(* IEC 61131-3 sources: moqui-plc/iec61131/moqui/framework/src/main/org/moqui/util, 39 files *)

(* ---- Clocks.dut ---- *)
(*#-#-#-#-#-#-#-#-#-#---Declaration---#-#-#-#-#-#-#-#-#-#-#-#-#*)

(* Generated clocks for timing generation *)
TYPE Clocks : STRUCT
	(*
     * SystemClock is the main high-speed clock, e.g., from the task cycle.
     * All other clocks are derived from it.
     *)
    systemClock : BOOL; (* Main system clock 100 Hz, duty-cycle 50% *)
    (* Derived clock pulses (one-cycle TRUE). Derived from systemClock rising edge *)
    clock10ms : BOOL; (* 10ms pulse *)
    clock100ms : BOOL; (* 100ms pulse *)
    clock1s : BOOL; (* 1 second pulse *)
    clock1minute : BOOL; (* 1 minute pulse *)
	(* Extend based on your needs *)
END_STRUCT END_TYPE

(* ---- Clocks.st ---- *)
(* Generated clocks for timing generation *)
TYPE Clocks : STRUCT
	(*
     * SystemClock is the main high-speed clock, e.g., from the task cycle.
     * All other clocks are derived from it.
     *)
    systemClock : BOOL; (* Main system clock 100 Hz, duty-cycle 50% *)
    (* Derived clock pulses (one-cycle TRUE). Derived from systemClock rising edge *)
    clock10ms : BOOL; (* 10ms pulse *)
    clock100ms : BOOL; (* 100ms pulse *)
    clock1s : BOOL; (* 1 second pulse *)
    clock1minute : BOOL; (* 1 minute pulse *)
	(* Extend based on your needs *)
END_STRUCT END_TYPE

(* ---- MeanFilterType.dut ---- *)
(*#-#-#-#-#-#-#-#-#-#---Declaration---#-#-#-#-#-#-#-#-#-#-#-#-#*)

{attribute 'qualified_only'}
{attribute 'strict'}
TYPE MeanFilterType : (
    SMA, (* Simple Moving Average *)
    WMA_Ramp, (* Weighted Moving Average, linear weights 1..N from oldest..newest (O(1)) *)
    WMA_Triangular, (* Symmetric triangular weights, center-weighted (O(N)) *)
    WMA_TriangularOddOnly, (* Symmetric triangular weights, requires odd windowSize (O(N)) *)
    TRI_SMA2, (* Triangular approximation via two SMA in cascade (O(1) per tick, extra memory) *)
    EMA (* Exponential Moving Average (alpha mandatory) *)
); END_TYPE

(* ---- doubleWordToReal.pou ---- *)
(*#-#-#-#-#-#-#-#-#-#---Declaration---#-#-#-#-#-#-#-#-#-#-#-#-#*)

(* Utility function to convert a word array to a real variable *)
FUNCTION doubleWordToReal : REAL
VAR_INPUT
	wordArray : ARRAY[0..1] OF WORD;
	bigEndian : BOOL := FALSE;
END_VAR
VAR
    dwordValue : DWORD;
END_VAR

(*#-#-#-#-#-#-#-#-#-#---Implementation---#-#-#-#-#-#-#-#-#-#-#-#-#*)

dwordValue := SHL(TO_DWORD(wordArray[0]), 16) OR TO_DWORD(wordArray[1]);
IF bigEndian THEN
    dwordValue := swapDWordEndian(dwordValue);
END_IF;
doubleWordToReal := TO_REAL(dwordValue);

(* ---- doubleWordToReal.st ---- *)
(* Utility function to convert a word array to a real variable *)
FUNCTION doubleWordToReal : REAL
	VAR_INPUT
		wordArray : ARRAY[0..1] OF WORD;
		bigEndian : BOOL := FALSE;
	END_VAR
	VAR
	    dwordValue : DWORD;
	END_VAR

	dwordValue := SHL(TO_DWORD(wordArray[0]), 16) OR TO_DWORD(wordArray[1]);
	IF bigEndian THEN
	    dwordValue := swapDWordEndian(dwordValue);
	END_IF;
	doubleWordToReal := TO_REAL(dwordValue);
	END_FUNCTION

(* ---- longRealToWordArray.pou ---- *)
(*#-#-#-#-#-#-#-#-#-#---Declaration---#-#-#-#-#-#-#-#-#-#-#-#-#*)

(* Convert a long real variable to a word array *)
FUNCTION longRealToWordArray : ARRAY[0..3] OF WORD
VAR_INPUT
    value : LREAL;
    bigEndian : BOOL := FALSE;
END_VAR
VAR
    lwordValue : LWORD;
    result : ARRAY[0..3] OF WORD;
END_VAR

(*#-#-#-#-#-#-#-#-#-#---Implementation---#-#-#-#-#-#-#-#-#-#-#-#-#*)

lwordValue := TO_LWORD(value);
IF bigEndian THEN
    lwordValue := swapLWordEndian(lwordValue);
END_IF;

result[0] := TO_WORD(SHR(lwordValue, 48));
result[1] := TO_WORD(SHR(lwordValue, 32) AND 16#FFFF);
result[2] := TO_WORD(SHR(lwordValue, 16) AND 16#FFFF);
result[3] := TO_WORD(lwordValue AND 16#FFFF);
longRealToWordArray := result;

(* ---- longRealToWordArray.st ---- *)
(* Convert a long real variable to a word array *)
FUNCTION longRealToWordArray : ARRAY[0..3] OF WORD
	VAR_INPUT
	    value : LREAL;
	    bigEndian : BOOL := FALSE;
	END_VAR
	VAR
	    lwordValue : LWORD;
	    result : ARRAY[0..3] OF WORD;
	END_VAR

	lwordValue := TO_LWORD(value);
	IF bigEndian THEN
	    lwordValue := swapLWordEndian(lwordValue);
	END_IF;

	result[0] := TO_WORD(SHR(lwordValue, 48));
	result[1] := TO_WORD(SHR(lwordValue, 32) AND 16#FFFF);
	result[2] := TO_WORD(SHR(lwordValue, 16) AND 16#FFFF);
	result[3] := TO_WORD(lwordValue AND 16#FFFF);
	longRealToWordArray := result;
	END_FUNCTION

(* ---- longWordToLongReal.pou ---- *)
(*#-#-#-#-#-#-#-#-#-#---Declaration---#-#-#-#-#-#-#-#-#-#-#-#-#*)

(* Utility function to convert a word array to a long real variable *)
FUNCTION longWordToLongReal : LREAL
VAR_INPUT
	wordArray : ARRAY[0..3] OF WORD;
	bigEndian : BOOL := FALSE;
END_VAR
VAR
	lwordValue : LWORD;
	w : ARRAY[0..3] OF WORD;
END_VAR

(*#-#-#-#-#-#-#-#-#-#---Implementation---#-#-#-#-#-#-#-#-#-#-#-#-#*)

IF bigEndian THEN
    w[0] := wordArray[3];
    w[1] := wordArray[2];
    w[2] := wordArray[1];
    w[3] := wordArray[0];
ELSE
    w := wordArray;
END_IF;

lwordValue := TO_LWORD(w[3]);
lwordValue := SHL(lwordValue, 16) OR TO_LWORD(w[2]);
lwordValue := SHL(lwordValue, 16) OR TO_LWORD(w[1]);
lwordValue := SHL(lwordValue, 16) OR TO_LWORD(w[0]);
longWordToLongReal := TO_LREAL(lwordValue);

(* ---- longWordToLongReal.st ---- *)
(* Utility function to convert a word array to a long real variable *)
FUNCTION longWordToLongReal : LREAL
	VAR_INPUT
		wordArray : ARRAY[0..3] OF WORD;
		bigEndian : BOOL := FALSE;
	END_VAR
	VAR
		lwordValue : LWORD;
		w : ARRAY[0..3] OF WORD;
	END_VAR

	IF bigEndian THEN
	    w[0] := wordArray[3];
	    w[1] := wordArray[2];
	    w[2] := wordArray[1];
	    w[3] := wordArray[0];
	ELSE
	    w := wordArray;
	END_IF;

	lwordValue := TO_LWORD(w[3]);
	lwordValue := SHL(lwordValue, 16) OR TO_LWORD(w[2]);
	lwordValue := SHL(lwordValue, 16) OR TO_LWORD(w[1]);
	lwordValue := SHL(lwordValue, 16) OR TO_LWORD(w[0]);
	longWordToLongReal := TO_LREAL(lwordValue);
	END_FUNCTION

(* ---- nowTimestamp.pou ---- *)
(*#-#-#-#-#-#-#-#-#-#---Declaration---#-#-#-#-#-#-#-#-#-#-#-#-#*)

FUNCTION nowTimestamp : DATE_AND_TIME
VAR
    utcTimestamp: UDINT;
    localTimestamp: UDINT;
    result: SysTimeRtc.RTS_IEC_RESULT;
	nowTimestampLocalString : STRING;
END_VAR

(*#-#-#-#-#-#-#-#-#-#---Implementation---#-#-#-#-#-#-#-#-#-#-#-#-#*)

(* Get current UTC time *)
utcTimestamp := SysTimeRtcGet(result);
(* Handle error (log it, return a default timestamp, etc.) *)
IF result <> 0 THEN RETURN; END_IF;
(* Convert UTC seconds to local time *)
result := SysTimeRtcConvertUtcToLocal(utcTimestamp, localTimestamp);
IF result <> 0 THEN RETURN; END_IF;
(* Convert local time to data and time format *)
nowTimestamp := TO_DT(localTimestamp);
(* Convert date and time format to a string *)
nowTimestampLocalString := TO_STRING(nowTimestamp);

(* ---- nowTimestamp.st ---- *)
FUNCTION nowTimestamp : DATE_AND_TIME
	VAR
	    utcTimestamp: UDINT;
	    localTimestamp: UDINT;
	    result: SysTimeRtc.RTS_IEC_RESULT;
		nowTimestampLocalString : STRING;
	END_VAR

	(* Get current UTC time *)
	utcTimestamp := SysTimeRtcGet(result);
	(* Handle error (log it, return a default timestamp, etc.) *)
	IF result <> 0 THEN RETURN; END_IF;
	(* Convert UTC seconds to local time *)
	result := SysTimeRtcConvertUtcToLocal(utcTimestamp, localTimestamp);
	IF result <> 0 THEN RETURN; END_IF;
	(* Convert local time to data and time format *)
	nowTimestamp := TO_DT(localTimestamp);
	(* Convert date and time format to a string *)
	nowTimestampLocalString := TO_STRING(nowTimestamp);
	END_FUNCTION

(* ---- realToWordArray.pou ---- *)
(*#-#-#-#-#-#-#-#-#-#---Declaration---#-#-#-#-#-#-#-#-#-#-#-#-#*)

(* Convert a real variable to a word array *)
FUNCTION realToWordArray : ARRAY[0..1] OF WORD
VAR_INPUT
    value : REAL;
    bigEndian : BOOL := FALSE;
END_VAR
VAR
    dwordValue : DWORD;
    result : ARRAY[0..1] OF WORD;
END_VAR

(*#-#-#-#-#-#-#-#-#-#---Implementation---#-#-#-#-#-#-#-#-#-#-#-#-#*)

dwordValue := TO_DWORD(value);
IF bigEndian THEN
    dwordValue := swapDWordEndian(dwordValue);
END_IF;
result[0] := TO_WORD(SHR(dwordValue, 16));
result[1] := TO_WORD(dwordValue AND 16#FFFF);
realToWordArray := result;

(* ---- realToWordArray.st ---- *)
(* Convert a real variable to a word array *)
FUNCTION realToWordArray : ARRAY[0..1] OF WORD
	VAR_INPUT
	    value : REAL;
	    bigEndian : BOOL := FALSE;
	END_VAR
	VAR
	    dwordValue : DWORD;
	    result : ARRAY[0..1] OF WORD;
	END_VAR

	dwordValue := TO_DWORD(value);
	IF bigEndian THEN
	    dwordValue := swapDWordEndian(dwordValue);
	END_IF;
	result[0] := TO_WORD(SHR(dwordValue, 16));
	result[1] := TO_WORD(dwordValue AND 16#FFFF);
	realToWordArray := result;
	END_FUNCTION

(* ---- round.pou ---- *)
(*#-#-#-#-#-#-#-#-#-#---Declaration---#-#-#-#-#-#-#-#-#-#-#-#-#*)

FUNCTION round : REAL
VAR_INPUT
    inputValue : REAL;
    decimals : INT;
END_VAR
VAR
    factor : REAL;
    tempValue : REAL;
END_VAR

(*#-#-#-#-#-#-#-#-#-#---Implementation---#-#-#-#-#-#-#-#-#-#-#-#-#*)

factor := TO_REAL(EXP(LN(10.0) * decimals));
tempValue := inputValue * factor;

IF tempValue >= 0 THEN
    round := TO_REAL(TRUNC(tempValue + 0.5)) / factor;
ELSE
    round := TO_REAL(TRUNC(tempValue - 0.5)) / factor;
END_IF;

(* ---- round.st ---- *)
FUNCTION round : REAL
	VAR_INPUT
	    inputValue : REAL;
	    decimals : INT;
	END_VAR
	VAR
	    factor : REAL;
	    tempValue : REAL;
	END_VAR

	factor := TO_REAL(EXP(LN(10.0) * decimals));
	tempValue := inputValue * factor;

	IF tempValue >= 0 THEN
	    round := TO_REAL(TRUNC(tempValue + 0.5)) / factor;
	ELSE
	    round := TO_REAL(TRUNC(tempValue - 0.5)) / factor;
	END_IF;
	END_FUNCTION

(* ---- scale.pou ---- *)
(*#-#-#-#-#-#-#-#-#-#---Declaration---#-#-#-#-#-#-#-#-#-#-#-#-#*)

FUNCTION scale : REAL
VAR_INPUT
	inputValue: REAL;
	minInputValue: REAL;
	maxInputValue: REAL;
	minOutputValue: REAL;
	maxOutputValue: REAL;
END_VAR
VAR
	outputValue: REAL;
END_VAR

(*#-#-#-#-#-#-#-#-#-#---Implementation---#-#-#-#-#-#-#-#-#-#-#-#-#*)

IF maxInputValue <= minInputValue THEN
	outputValue := minOutputValue;
ELSE
    outputValue := (maxOutputValue - minOutputValue) / (maxInputValue - minInputValue)
		* (LIMIT(minInputValue, inputValue, maxInputValue) - minInputValue) + minOutputValue;
END_IF;
scale := outputValue;

(* ---- scale.st ---- *)
FUNCTION scale : REAL
	VAR_INPUT
		inputValue: REAL;
		minInputValue: REAL;
		maxInputValue: REAL;
		minOutputValue: REAL;
		maxOutputValue: REAL;
	END_VAR
	VAR
		outputValue: REAL;
	END_VAR

	IF maxInputValue <= minInputValue THEN
		outputValue := minOutputValue;
	ELSE
	    outputValue := (maxOutputValue - minOutputValue) / (maxInputValue - minInputValue)
			* (LIMIT(minInputValue, inputValue, maxInputValue) - minInputValue) + minOutputValue;
	END_IF;
	scale := outputValue;
	END_FUNCTION

(* ---- swapDWordEndian.pou ---- *)
(*#-#-#-#-#-#-#-#-#-#---Declaration---#-#-#-#-#-#-#-#-#-#-#-#-#*)

(* Swap two words in a double word to change the endianness *)
FUNCTION swapDWordEndian : DWORD
VAR_INPUT
    input : DWORD;
END_VAR

(*#-#-#-#-#-#-#-#-#-#---Implementation---#-#-#-#-#-#-#-#-#-#-#-#-#*)

swapDWordEndian := SHL(input AND 16#0000FFFF, 16) OR SHR(input AND 16#FFFF0000, 16);

(* ---- swapDWordEndian.st ---- *)
(* Swap two words in a double word to change the endianness *)
FUNCTION swapDWordEndian : DWORD
	VAR_INPUT
	    input : DWORD;
	END_VAR

	swapDWordEndian := SHL(input AND 16#0000FFFF, 16) OR SHR(input AND 16#FFFF0000, 16);
	END_FUNCTION

(* ---- swapLWordEndian.pou ---- *)
(*#-#-#-#-#-#-#-#-#-#---Declaration---#-#-#-#-#-#-#-#-#-#-#-#-#*)

(* Swap four words in an long word *)
FUNCTION swapLWordEndian : LWORD
VAR_INPUT
    input : LWORD;
END_VAR
VAR
    w0, w1, w2, w3 : WORD;
    result : LWORD;
END_VAR

(*#-#-#-#-#-#-#-#-#-#---Implementation---#-#-#-#-#-#-#-#-#-#-#-#-#*)

w0 := TO_WORD(SHR(input, 48));
w1 := TO_WORD(SHR(input, 32) AND 16#FFFF);
w2 := TO_WORD(SHR(input, 16) AND 16#FFFF);
w3 := TO_WORD(input AND 16#FFFF);
result := TO_LWORD(w3);
result := SHL(result, 16) OR TO_LWORD(w2);
result := SHL(result, 16) OR TO_LWORD(w1);
result := SHL(result, 16) OR TO_LWORD(w0);
swapLWordEndian := result;

(* ---- swapLWordEndian.st ---- *)
(* Swap four words in an long word *)
FUNCTION swapLWordEndian : LWORD
	VAR_INPUT
	    input : LWORD;
	END_VAR
	VAR
	    w0, w1, w2, w3 : WORD;
	    result : LWORD;
	END_VAR

	w0 := TO_WORD(SHR(input, 48));
	w1 := TO_WORD(SHR(input, 32) AND 16#FFFF);
	w2 := TO_WORD(SHR(input, 16) AND 16#FFFF);
	w3 := TO_WORD(input AND 16#FFFF);
	result := TO_LWORD(w3);
	result := SHL(result, 16) OR TO_LWORD(w2);
	result := SHL(result, 16) OR TO_LWORD(w1);
	result := SHL(result, 16) OR TO_LWORD(w0);
	swapLWordEndian := result;
	END_FUNCTION

(* ---- swapWordEndian.pou ---- *)
(*#-#-#-#-#-#-#-#-#-#---Declaration---#-#-#-#-#-#-#-#-#-#-#-#-#*)

(* Swap bytes in a word to change the endianness *)
FUNCTION swapWordEndian : WORD
VAR_INPUT
    input : WORD;
END_VAR

(*#-#-#-#-#-#-#-#-#-#---Implementation---#-#-#-#-#-#-#-#-#-#-#-#-#*)

swapWordEndian := SHL(input AND 16#00FF, 8) OR SHR(input AND 16#FF00, 8);

(* ---- swapWordEndian.st ---- *)
(* Swap bytes in a word to change the endianness *)
FUNCTION swapWordEndian : WORD
	VAR_INPUT
	    input : WORD;
	END_VAR

	swapWordEndian := SHL(input AND 16#00FF, 8) OR SHR(input AND 16#FF00, 8);
	END_FUNCTION

(* ---- toByteArray.pou ---- *)
(*#-#-#-#-#-#-#-#-#-#---Declaration---#-#-#-#-#-#-#-#-#-#-#-#-#*)

FUNCTION toByteArray : BOOL
VAR_INPUT
    inputWord : WORD;
END_VAR
VAR_OUTPUT
	byteArray : ARRAY [0..1] OF BYTE; (* Output array: [highByte, lowByte] *)
END_VAR

(*#-#-#-#-#-#-#-#-#-#---Implementation---#-#-#-#-#-#-#-#-#-#-#-#-#*)

toByteArray := FALSE;
(* Extract high and low byte *)
byteArray[0] := TO_BYTE(SHR(inputWord, 8)); (* High byte *)
byteArray[1] := TO_BYTE(inputWord AND 16#00FF); (* Low byte *)
toByteArray := TRUE;

(* ---- toByteArray.st ---- *)
FUNCTION toByteArray : BOOL
	VAR_INPUT
	    inputWord : WORD;
	END_VAR
	VAR_OUTPUT
		byteArray : ARRAY [0..1] OF BYTE; (* Output array: [highByte, lowByte] *)
	END_VAR

	toByteArray := FALSE;
	(* Extract high and low byte *)
	byteArray[0] := TO_BYTE(SHR(inputWord, 8)); (* High byte *)
	byteArray[1] := TO_BYTE(inputWord AND 16#00FF); (* Low byte *)
	toByteArray := TRUE;
	END_FUNCTION

(* ---- trim.pou ---- *)
(*#-#-#-#-#-#-#-#-#-#---Declaration---#-#-#-#-#-#-#-#-#-#-#-#-#*)

FUNCTION trim : STRING
VAR_INPUT
    inputString : STRING;
END_VAR
VAR
    startPos, endPos : INT;
    stringLength : INT;
    currentCharCode : INT;
END_VAR

(*#-#-#-#-#-#-#-#-#-#---Implementation---#-#-#-#-#-#-#-#-#-#-#-#-#*)

stringLength := LEN(inputString);
startPos := 1;

(* Skip leading whitespace (space, tab = 9, LF = 10, CR = 13) *)
WHILE (startPos <= stringLength) DO
    currentCharCode := TO_INT(MID(inputString, startPos, 1));
    IF (currentCharCode <> 32) AND (currentCharCode <> 9)
			AND (currentCharCode <> 10) AND (currentCharCode <> 13) THEN
        EXIT;
    END_IF;

    startPos := startPos + 1;
END_WHILE;

(* Skip trailing whitespace *)
endPos := stringLength;
WHILE (endPos > 0) DO
    currentCharCode := TO_INT(MID(inputString, endPos, 1));
    IF (currentCharCode <> 32) AND (currentCharCode <> 9)
			AND (currentCharCode <> 10) AND (currentCharCode <> 13) THEN
        EXIT;
    END_IF;

    endPos := endPos - 1;
END_WHILE;

(* Extract the trimmed substring *)
IF startPos <= endPos THEN
    trim := MID(inputString, startPos, endPos - startPos + 1);
ELSE
    trim := ''; (* All characters were whitespace *)
END_IF;

(* ---- trim.st ---- *)
FUNCTION trim : STRING
	VAR_INPUT
	    inputString : STRING;
	END_VAR
	VAR
	    startPos, endPos : INT;
	    stringLength : INT;
	    currentCharCode : INT;
	END_VAR

	stringLength := LEN(inputString);
	startPos := 1;

	(* Skip leading whitespace (space, tab = 9, LF = 10, CR = 13) *)
	WHILE (startPos <= stringLength) DO
	    currentCharCode := TO_INT(MID(inputString, startPos, 1));
	    IF (currentCharCode <> 32) AND (currentCharCode <> 9)
				AND (currentCharCode <> 10) AND (currentCharCode <> 13) THEN
	        EXIT;
	    END_IF;

	    startPos := startPos + 1;
	END_WHILE;

	(* Skip trailing whitespace *)
	endPos := stringLength;
	WHILE (endPos > 0) DO
	    currentCharCode := TO_INT(MID(inputString, endPos, 1));
	    IF (currentCharCode <> 32) AND (currentCharCode <> 9)
				AND (currentCharCode <> 10) AND (currentCharCode <> 13) THEN
	        EXIT;
	    END_IF;

	    endPos := endPos - 1;
	END_WHILE;

	(* Extract the trimmed substring *)
	IF startPos <= endPos THEN
	    trim := MID(inputString, startPos, endPos - startPos + 1);
	ELSE
	    trim := ''; (* All characters were whitespace *)
	END_IF;
	END_FUNCTION

(* ---- truncReal.pou ---- *)
(*#-#-#-#-#-#-#-#-#-#---Declaration---#-#-#-#-#-#-#-#-#-#-#-#-#*)

FUNCTION truncReal : REAL
VAR_INPUT
    inputValue : REAL;
    decimals : INT;
END_VAR
VAR
    factor : REAL;
END_VAR

(*#-#-#-#-#-#-#-#-#-#---Implementation---#-#-#-#-#-#-#-#-#-#-#-#-#*)

factor := TO_REAL(EXP(LN(10.0) * TO_REAL(decimals)));
truncReal := TO_REAL(TRUNC(inputValue * factor)) / factor;

(* ---- truncReal.st ---- *)
FUNCTION truncReal : REAL
	VAR_INPUT
	    inputValue : REAL;
	    decimals : INT;
	END_VAR
	VAR
	    factor : REAL;
	END_VAR

	factor := TO_REAL(EXP(LN(10.0) * TO_REAL(decimals)));
	truncReal := TO_REAL(TRUNC(inputValue * factor)) / factor;
	END_FUNCTION

(* ---- ClockGeneration.pou ---- *)
(*#-#-#-#-#-#-#-#-#-#---Declaration---#-#-#-#-#-#-#-#-#-#-#-#-#*)

{attribute 'no_assign'}
(* Timing generation *)
FUNCTION_BLOCK ClockGeneration
VAR_EXTERNAL
	clks : Clocks;
END_VAR
VAR_INPUT
	operationType : OperatingMode;
END_VAR
VAR
	(* Internal variable to detect the rising edge of the systemClock *)
	systemClockOld : BOOL;
	(* Internal counters for derived clocks *)
	timerClock100ms : UDINT;
	timerClock1s : UDINT;
	timerClock1minute : UDINT;
END_VAR

(*#-#-#-#-#-#-#-#-#-#---Implementation---#-#-#-#-#-#-#-#-#-#-#-#-#*)

IF (operationType = OperatingMode.Init) THEN
	systemClockOld := TRUE;
	timerClock100ms := 10;
	timerClock1s := 10;
	timerClock1minute := 60;
END_IF;

(*
 * Uncomment if you want to make loops shorter than 10 ms.
 * It is not recommended to go below 5 ms with the PLC.
 * The control loop (current) of the axes is in the servo drives.
 *)
(*
clks.clock10ms := clks.systemClock AND NOT systemClockOld;
systemClockOld := clks.systemClock;
*)
clks.clock10ms := TRUE;

IF clks.clock10ms THEN
	timerClock100ms := timerClock100ms - 1;
END_IF;
clks.clock100ms := (timerClock100ms = 0);

IF clks.clock100ms THEN
	timerClock100ms := 10;
	timerClock1s := timerClock1s - 1;
END_IF;
clks.clock1s := (timerClock1s = 0);

IF clks.clock1s THEN
	timerClock1s := 10;
	timerClock1minute := timerClock1minute - 1;
END_IF;
clks.clock1minute := (timerClock1minute = 0);

IF clks.clock1minute THEN
	timerClock1minute := 60;
END_IF;

(* ---- ClockGeneration.st ---- *)
(* Timing generation *)
FUNCTION_BLOCK ClockGeneration
	VAR_EXTERNAL
		clks : Clocks;
	END_VAR
	VAR_INPUT
		operationType : OperatingMode;
	END_VAR
	VAR
		(* Internal variable to detect the rising edge of the systemClock *)
		systemClockOld : BOOL;
		(* Internal counters for derived clocks *)
		timerClock100ms : UDINT;
		timerClock1s : UDINT;
		timerClock1minute : UDINT;
	END_VAR

	IF (operationType = OperatingMode.Init) THEN
		systemClockOld := TRUE;
		timerClock100ms := 10;
		timerClock1s := 10;
		timerClock1minute := 60;
	END_IF;

	(*
	 * Uncomment if you want to make loops shorter than 10 ms.
	 * It is not recommended to go below 5 ms with the PLC.
	 * The control loop (current) of the axes is in the servo drives.
	 *)
	(*
	clks.clock10ms := clks.systemClock AND NOT systemClockOld;
	systemClockOld := clks.systemClock;
	*)
	clks.clock10ms := TRUE;

	IF clks.clock10ms THEN
		timerClock100ms := timerClock100ms - 1;
	END_IF;
	clks.clock100ms := (timerClock100ms = 0);

	IF clks.clock100ms THEN
		timerClock100ms := 10;
		timerClock1s := timerClock1s - 1;
	END_IF;
	clks.clock1s := (timerClock1s = 0);

	IF clks.clock1s THEN
		timerClock1s := 10;
		timerClock1minute := timerClock1minute - 1;
	END_IF;
	clks.clock1minute := (timerClock1minute = 0);

	IF clks.clock1minute THEN
		timerClock1minute := 60;
	END_IF;
	END_FUNCTION_BLOCK

(* ---- Filter.pou ---- *)
(*#-#-#-#-#-#-#-#-#-#---Declaration---#-#-#-#-#-#-#-#-#-#-#-#-#*)

(* Signal filtering and deboucing.
   Usage:

       (* heatingPlatesOpened *)
       VAR
           heatingPlatesOpenedFilter : Filter;
       END_VAR

       heatingPlatesOpenedFilter(operationType := operationType, clock := heatingPlatesControlClock,
           signal := heatingPlatesOpened, activationDelay := 0, deactivationDelay := heatingPlatesOpeningDelay,
	   	   delayedSignal => heatingPlatesOpened);
 *)
FUNCTION_BLOCK Filter
VAR_INPUT
	operationType : OperatingMode;
	clock : BOOL;
	signal : BOOL;
	activationDelay : UDINT;
	deactivationDelay : UDINT;
END_VAR
VAR_OUTPUT
	delayedSignal : BOOL;
END_VAR
VAR
	delay : UDINT;
END_VAR

(*#-#-#-#-#-#-#-#-#-#---Implementation---#-#-#-#-#-#-#-#-#-#-#-#-#*)

IF (operationType = OperatingMode.Init) THEN
	delay := 0;
END_IF;

IF clock AND (delay > 0) THEN
	delay := delay - 1;
END_IF;

IF delay = 0 THEN
	delayedSignal := signal;
END_IF;

IF signal = delayedSignal THEN
	IF signal THEN
		delay := deactivationDelay;
	ELSE
		delay := activationDelay;
	END_IF;
END_IF;

(* ---- Filter.st ---- *)
(* Signal filtering and deboucing.
   Usage:

       (* heatingPlatesOpened *)
       VAR
           heatingPlatesOpenedFilter : Filter;
       END_VAR

       heatingPlatesOpenedFilter(operationType := operationType, clock := heatingPlatesControlClock,
           signal := heatingPlatesOpened, activationDelay := 0, deactivationDelay := heatingPlatesOpeningDelay,
	   	   delayedSignal => heatingPlatesOpened);
 *)
FUNCTION_BLOCK Filter
VAR_INPUT
	operationType : OperatingMode;
	clock : BOOL;
	signal : BOOL;
	activationDelay : UDINT;
	deactivationDelay : UDINT;
END_VAR
VAR_OUTPUT
	delayedSignal : BOOL;
END_VAR
VAR
	delay : UDINT;
END_VAR

IF (operationType = OperatingMode.Init) THEN
	delay := 0;
END_IF;

IF clock AND (delay > 0) THEN
	delay := delay - 1;
END_IF;

IF delay = 0 THEN
	delayedSignal := signal;
END_IF;

IF signal = delayedSignal THEN
	IF signal THEN
		delay := deactivationDelay;
	ELSE
		delay := activationDelay;
	END_IF;
END_IF;

(* ---- IIRFilter.pou ---- *)
(*#-#-#-#-#-#-#-#-#-#---Declaration---#-#-#-#-#-#-#-#-#-#-#-#-#*)

{attribute 'no_assign'}
FUNCTION_BLOCK IIRFilter
VAR_INPUT
    execute : BOOL;
    clock : BOOL;
    reset : BOOL;
    input : REAL;
    T : REAL; (* Time constant in seconds *)
    tickTime : TIME := T#10ms; (* Sampling period *)
END_VAR
VAR_OUTPUT
    output : REAL;
    done : BOOL;
    busy : BOOL;
    error : BOOL;
    errorId : INT; (* 1 : InvalidTime *)
    timeElapsed : REAL; (* Time elapsed in seconds *)
END_VAR
VAR
    init : BOOL;
    elapsedTicks : UDINT;
    deltaTime : REAL;
    alpha : REAL;
END_VAR

(*#-#-#-#-#-#-#-#-#-#---Implementation---#-#-#-#-#-#-#-#-#-#-#-#-#*)

(* Defaults *)
done := FALSE; busy := FALSE; error := FALSE; errorId := 0;

(* Validate tickTime *)
IF TO_DINT(tickTime) <= 0 THEN
    error := execute;
    errorId := 1;
    busy := FALSE;
    RETURN;
END_IF;

deltaTime := TO_REAL(TO_DINT(tickTime)) / 1000.0; (* seconds per tick *)

IF reset THEN
    init := FALSE;
    elapsedTicks := 0;
END_IF;

IF execute THEN
    busy := TRUE;

    (* Initialize output to current input on first enable *)
    IF NOT init THEN
        output := input;
        init := TRUE;
        elapsedTicks := 0;
    ELSE
        (* Update only on external tick *)
        IF clock THEN
            (* alpha = 1 - exp(-dt/T) *)
            IF T > 0.0 THEN
                alpha := 1.0 - EXP(-deltaTime / T);
                output := output + alpha * (input - output);
            ELSE
                output := input;
            END_IF;

            elapsedTicks := elapsedTicks + 1;
        END_IF;
    END_IF;

    timeElapsed := TO_REAL(elapsedTicks) * deltaTime;

    done := NOT error;
ELSE
    busy := FALSE;
    done := FALSE;
    timeElapsed := 0.0;
END_IF;

(* ---- IIRFilter.st ---- *)
FUNCTION_BLOCK IIRFilter
	VAR_INPUT
	    execute : BOOL;
	    clock : BOOL;
	    reset : BOOL;
	    input : REAL;
	    T : REAL; (* Time constant in seconds *)
	    tickTime : TIME := T#10ms; (* Sampling period *)
	END_VAR
	VAR_OUTPUT
	    output : REAL;
	    done : BOOL;
	    busy : BOOL;
	    error : BOOL;
	    errorId : INT; (* 1 : InvalidTime *)
	    timeElapsed : REAL; (* Time elapsed in seconds *)
	END_VAR
	VAR
	    init : BOOL;
	    elapsedTicks : UDINT;
	    deltaTime : REAL;
	    alpha : REAL;
	END_VAR

	(* Defaults *)
	done := FALSE; busy := FALSE; error := FALSE; errorId := 0;

	(* Validate tickTime *)
	IF TO_DINT(tickTime) <= 0 THEN
	    error := execute;
	    errorId := 1;
	    busy := FALSE;
	    RETURN;
	END_IF;

	deltaTime := TO_REAL(TO_DINT(tickTime)) / 1000.0; (* seconds per tick *)

	IF reset THEN
	    init := FALSE;
	    elapsedTicks := 0;
	END_IF;

	IF execute THEN
	    busy := TRUE;

	    (* Initialize output to current input on first enable *)
	    IF NOT init THEN
	        output := input;
	        init := TRUE;
	        elapsedTicks := 0;
	    ELSE
	        (* Update only on external tick *)
	        IF clock THEN
	            (* alpha = 1 - exp(-dt/T) *)
	            IF T > 0.0 THEN
	                alpha := 1.0 - EXP(-deltaTime / T);
	                output := output + alpha * (input - output);
	            ELSE
	                output := input;
	            END_IF;

	            elapsedTicks := elapsedTicks + 1;
	        END_IF;
	    END_IF;

	    timeElapsed := TO_REAL(elapsedTicks) * deltaTime;

	    done := NOT error;
	ELSE
	    busy := FALSE;
	    done := FALSE;
	    timeElapsed := 0.0;
	END_IF;
	END_FUNCTION_BLOCK

(* ---- MeanFilter.pou ---- *)
(*#-#-#-#-#-#-#-#-#-#---Declaration---#-#-#-#-#-#-#-#-#-#-#-#-#*)

{attribute 'no_assign'}
(* Mean / Moving Average Filter: SMA, WMA_Ramp, WMA_Triangular(+OddOnly), TRI_SMA2, EMA *)
FUNCTION_BLOCK MeanFilter
VAR_INPUT
    execute : BOOL; (* Enable filter *)
    clock : BOOL;   (* Tick pulse (one-scan TRUE) *)
    reset : BOOL;
    input : REAL;

    filterType : MeanFilterType := MeanFilterType.SMA;

    (* Windowed filters (SMA/WMA) *)
    windowSize : UINT := 10; (* must be <= MAX_WINDOW *)

    (* EMA parameters (alpha mandatory) *)
    emaAlpha : REAL := 0.1; (* MUST be in (0..1] *)
END_VAR
VAR_OUTPUT
    output : REAL;
    done : BOOL;
    busy : BOOL;
    error : BOOL;
    errorId : INT; (* 1: InvalidWindow, 3: InvalidAlpha, 4: RequiresOddWindow *)
END_VAR
VAR CONSTANT
    MAX_WINDOW : UINT := 256;
END_VAR
VAR
    buffer : ARRAY[1..MAX_WINDOW] OF REAL;
    idx : UINT; (* Next position to overwrite = oldest sample *)
    initialized : BOOL;
    (* Common *)
    i : UINT;
    (* SMA *)
    sum : REAL;
    (* WMA_Ramp (linear 1..N) *)
    wsumRamp : REAL; (* Σ(k*x_k) *)
    denomRamp : REAL; (* N(N+1)/2 *)
    xOld : REAL;
    xNew : REAL;
    sumOld : REAL;
    (* WMA_Triangular *)
    wsumTri : REAL;
    denomTri : REAL;
    pos : UINT;
    w : REAL;
    k : UINT; (* 1..N position from oldest..newest *)
    mid : UINT; (* floor((N+1)/2) *)
    dist : UINT;
    (* TRI_SMA2 (two SMA in cascade) *)
    sma2_buf1 : ARRAY[1..MAX_WINDOW] OF REAL;
    sma2_buf2 : ARRAY[1..MAX_WINDOW] OF REAL;
    sma2_idx1 : UINT;
    sma2_idx2 : UINT;
    sma2_sum1 : REAL;
    sma2_sum2 : REAL;
    sma2_y1 : REAL;
    sma2_y2 : REAL;
    sma2_init : BOOL;
    (* EMA *)
    emaY : REAL;
    (* Config change detection *)
    prevType : MeanFilterType;
    prevWindow : UINT;
END_VAR

(*#-#-#-#-#-#-#-#-#-#---Implementation---#-#-#-#-#-#-#-#-#-#-#-#-#*)

done := FALSE; busy := FALSE; error := FALSE; errorId := 0;

(* Config change forces internal reset *)
IF (filterType <> prevType) OR (windowSize <> prevWindow) THEN
    reset := TRUE;
END_IF;
prevType := filterType;
prevWindow := windowSize;

CASE filterType OF
	(* Validate window for windowed filters *)
	MeanFilterType.SMA, MeanFilterType.WMA_Ramp,
   	MeanFilterType.WMA_Triangular, MeanFilterType.WMA_TriangularOddOnly,
	MeanFilterType.TRI_SMA2 :

		IF (windowSize = 0) OR (windowSize > MAX_WINDOW) THEN
			error := execute;
			errorId := 1;
			RETURN;
		END_IF;

		(* Odd-only constraint: checked here because CASE does not fall-through *)
		IF (filterType = MeanFilterType.WMA_TriangularOddOnly) AND ((windowSize MOD 2) = 0) THEN
			error := execute;
			errorId := 4;
			RETURN;
		END_IF;

	(* Validate alpha for EMA *)
	MeanFilterType.EMA :
		IF (emaAlpha <= 0.0) OR (emaAlpha > 1.0) THEN
			error := execute;
			errorId := 3;
			RETURN;
		END_IF;
END_CASE;

IF reset THEN
    idx := 1;
    initialized := FALSE;

    sum := 0.0;

    wsumRamp := 0.0;
    denomRamp := 0.0;

    wsumTri := 0.0;
    denomTri := 0.0;

    emaY := 0.0;

    sma2_idx1 := 1;
    sma2_idx2 := 1;
    sma2_sum1 := 0.0;
    sma2_sum2 := 0.0;
    sma2_y1 := 0.0;
    sma2_y2 := 0.0;
    sma2_init := FALSE;

    (* Optional: clear buffers *)
    FOR i := 1 TO MAX_WINDOW DO
        buffer[i] := 0.0;
        sma2_buf1[i] := 0.0;
        sma2_buf2[i] := 0.0;
    END_FOR;
END_IF;

IF execute THEN
    busy := TRUE;

    CASE filterType OF
        MeanFilterType.SMA :
            IF NOT initialized THEN
                (* Prime buffer with first input *)
                FOR i := 1 TO windowSize DO buffer[i] := input; END_FOR;
                sum := input * TO_REAL(windowSize);
                idx := 1;
                initialized := TRUE;
                output := input;
            ELSE
                IF clock THEN
                    xOld := buffer[idx];
                    buffer[idx] := input;

                    sum := sum - xOld + input;

                    idx := idx + 1;
                    IF idx > windowSize THEN idx := 1; END_IF;

                    output := sum / TO_REAL(windowSize);
                END_IF;
            END_IF;

        MeanFilterType.WMA_Ramp :
            (* Linear weights: 1..N from oldest..newest (O(1)) *)
            IF NOT initialized THEN
                FOR i := 1 TO windowSize DO buffer[i] := input; END_FOR;

                denomRamp := TO_REAL(windowSize) * TO_REAL(windowSize + 1) / 2.0;

                sum := input * TO_REAL(windowSize);
                wsumRamp := input * denomRamp;

                idx := 1;
                initialized := TRUE;
                output := input;
            ELSE
                IF clock THEN
                    xOld := buffer[idx]; (* oldest *)
                    xNew := input;

                    sumOld := sum;

                    buffer[idx] := xNew;

                    (* S' = S - xOld + xNew *)
                    sum := sumOld - xOld + xNew;

                    (* W' = W - S_old + N*xNew *)
                    wsumRamp := wsumRamp - sumOld + (TO_REAL(windowSize) * xNew);

                    idx := idx + 1;
                    IF idx > windowSize THEN idx := 1; END_IF;

                    output := wsumRamp / denomRamp;
                END_IF;
            END_IF;

        MeanFilterType.WMA_Triangular,
        MeanFilterType.WMA_TriangularOddOnly :
            (* Symmetric triangular weights, center-weighted (O(N)) *)
            IF NOT initialized THEN
                FOR i := 1 TO windowSize DO buffer[i] := input; END_FOR;
                idx := 1;
                initialized := TRUE;
                output := input;
            END_IF;

            IF clock THEN
                (* Update ring buffer *)
                buffer[idx] := input;
                idx := idx + 1;
                IF idx > windowSize THEN idx := 1; END_IF;

                (* Compute triangular weights *)
                (* k=1..N from oldest..newest *)
                mid := (windowSize + 1) / 2; (* integer div *)

                wsumTri := 0.0;
                denomTri := 0.0;

                (* Oldest sample is at idx (next to overwrite) *)
                FOR i := 0 TO windowSize - 1 DO
                    pos := idx + i;
                    IF pos > windowSize THEN pos := pos - windowSize; END_IF;

                    k := i + 1;

                    (* w = mid - |k-mid|  (triangle peak at center) *)
                    IF k >= mid THEN
                        dist := k - mid;
                    ELSE
                        dist := mid - k;
                    END_IF;

                    w := TO_REAL(mid - dist);
                    wsumTri := wsumTri + w * buffer[pos];
                    denomTri := denomTri + w;
                END_FOR;

                IF denomTri > 0.0 THEN
                    output := wsumTri / denomTri;
                ELSE
                    output := input;
                END_IF;
            END_IF;

        MeanFilterType.TRI_SMA2 :
            (*
             * Triangular approximation via two SMA in cascade:
             *     y1 = SMA(input), y2 = SMA(y1). This approximates a triangular FIR well.
            *)
            IF NOT sma2_init THEN
                FOR i := 1 TO windowSize DO
                    sma2_buf1[i] := input;
                    sma2_buf2[i] := input;
                END_FOR;

                sma2_sum1 := input * TO_REAL(windowSize);
                sma2_sum2 := input * TO_REAL(windowSize);

                sma2_idx1 := 1;
                sma2_idx2 := 1;

                sma2_y1 := input;
                sma2_y2 := input;

                sma2_init := TRUE;
                output := input;
            ELSE
                IF clock THEN
                    (* SMA stage 1 *)
                    xOld := sma2_buf1[sma2_idx1];
                    sma2_buf1[sma2_idx1] := input;
                    sma2_sum1 := sma2_sum1 - xOld + input;

                    sma2_idx1 := sma2_idx1 + 1;
                    IF sma2_idx1 > windowSize THEN sma2_idx1 := 1; END_IF;

                    sma2_y1 := sma2_sum1 / TO_REAL(windowSize);

                    (* SMA stage 2 *)
                    xOld := sma2_buf2[sma2_idx2];
                    sma2_buf2[sma2_idx2] := sma2_y1;
                    sma2_sum2 := sma2_sum2 - xOld + sma2_y1;

                    sma2_idx2 := sma2_idx2 + 1;
                    IF sma2_idx2 > windowSize THEN sma2_idx2 := 1; END_IF;

                    sma2_y2 := sma2_sum2 / TO_REAL(windowSize);

                    output := sma2_y2;
                END_IF;
            END_IF;

        MeanFilterType.EMA :
            (* EMA (alpha mandatory) *)
            IF NOT initialized THEN
                emaY := input;
                initialized := TRUE;
            ELSE
                IF clock THEN
                    emaY := emaY + emaAlpha * (input - emaY);
                END_IF;
            END_IF;

            output := emaY;
    END_CASE;

    done := NOT error;
ELSE
    busy := FALSE;
    done := FALSE;
END_IF;

(* ---- MeanFilter.st ---- *)
(* Mean / Moving Average Filter: SMA, WMA_Ramp, WMA_Triangular(+OddOnly), TRI_SMA2, EMA *)
FUNCTION_BLOCK MeanFilter
	VAR_INPUT
	    execute : BOOL; (* Enable filter *)
	    clock : BOOL;   (* Tick pulse (one-scan TRUE) *)
	    reset : BOOL;
	    input : REAL;

	    filterType : MeanFilterType := MeanFilterType.SMA;

	    (* Windowed filters (SMA/WMA) *)
	    windowSize : UINT := 10; (* must be <= MAX_WINDOW *)

	    (* EMA parameters (alpha mandatory) *)
	    emaAlpha : REAL := 0.1; (* MUST be in (0..1] *)
	END_VAR
	VAR_OUTPUT
	    output : REAL;
	    done : BOOL;
	    busy : BOOL;
	    error : BOOL;
	    errorId : INT; (* 1: InvalidWindow, 3: InvalidAlpha, 4: RequiresOddWindow *)
	END_VAR
	VAR CONSTANT
	    MAX_WINDOW : UINT := 256;
	END_VAR
	VAR
	    buffer : ARRAY[1..MAX_WINDOW] OF REAL;
	    idx : UINT; (* Next position to overwrite = oldest sample *)
	    initialized : BOOL;
	    (* Common *)
	    i : UINT;
	    (* SMA *)
	    sum : REAL;
	    (* WMA_Ramp (linear 1..N) *)
	    wsumRamp : REAL; (* Σ(k*x_k) *)
	    denomRamp : REAL; (* N(N+1)/2 *)
	    xOld : REAL;
	    xNew : REAL;
	    sumOld : REAL;
	    (* WMA_Triangular *)
	    wsumTri : REAL;
	    denomTri : REAL;
	    pos : UINT;
	    w : REAL;
	    k : UINT; (* 1..N position from oldest..newest *)
	    mid : UINT; (* floor((N+1)/2) *)
	    dist : UINT;
	    (* TRI_SMA2 (two SMA in cascade) *)
	    sma2_buf1 : ARRAY[1..MAX_WINDOW] OF REAL;
	    sma2_buf2 : ARRAY[1..MAX_WINDOW] OF REAL;
	    sma2_idx1 : UINT;
	    sma2_idx2 : UINT;
	    sma2_sum1 : REAL;
	    sma2_sum2 : REAL;
	    sma2_y1 : REAL;
	    sma2_y2 : REAL;
	    sma2_init : BOOL;
	    (* EMA *)
	    emaY : REAL;
	    (* Config change detection *)
	    prevType : MeanFilterType;
	    prevWindow : UINT;
	END_VAR

	done := FALSE; busy := FALSE; error := FALSE; errorId := 0;

	(* Config change forces internal reset *)
	IF (filterType <> prevType) OR (windowSize <> prevWindow) THEN
	    reset := TRUE;
	END_IF;
	prevType := filterType;
	prevWindow := windowSize;

	CASE filterType OF
		(* Validate window for windowed filters *)
		MeanFilterType.SMA, MeanFilterType.WMA_Ramp,
	   	MeanFilterType.WMA_Triangular, MeanFilterType.WMA_TriangularOddOnly,
		MeanFilterType.TRI_SMA2 :

			IF (windowSize = 0) OR (windowSize > MAX_WINDOW) THEN
				error := execute;
				errorId := 1;
				RETURN;
			END_IF;

			(* Odd-only constraint: checked here because CASE does not fall-through *)
			IF (filterType = MeanFilterType.WMA_TriangularOddOnly) AND ((windowSize MOD 2) = 0) THEN
				error := execute;
				errorId := 4;
				RETURN;
			END_IF;

		(* Validate alpha for EMA *)
		MeanFilterType.EMA :
			IF (emaAlpha <= 0.0) OR (emaAlpha > 1.0) THEN
				error := execute;
				errorId := 3;
				RETURN;
			END_IF;
	END_CASE;

	IF reset THEN
	    idx := 1;
	    initialized := FALSE;

	    sum := 0.0;

	    wsumRamp := 0.0;
	    denomRamp := 0.0;

	    wsumTri := 0.0;
	    denomTri := 0.0;

	    emaY := 0.0;

	    sma2_idx1 := 1;
	    sma2_idx2 := 1;
	    sma2_sum1 := 0.0;
	    sma2_sum2 := 0.0;
	    sma2_y1 := 0.0;
	    sma2_y2 := 0.0;
	    sma2_init := FALSE;

	    (* Optional: clear buffers *)
	    FOR i := 1 TO MAX_WINDOW DO
	        buffer[i] := 0.0;
	        sma2_buf1[i] := 0.0;
	        sma2_buf2[i] := 0.0;
	    END_FOR;
	END_IF;

	IF execute THEN
	    busy := TRUE;

	    CASE filterType OF
	        MeanFilterType.SMA :
	            IF NOT initialized THEN
	                (* Prime buffer with first input *)
	                FOR i := 1 TO windowSize DO buffer[i] := input; END_FOR;
	                sum := input * TO_REAL(windowSize);
	                idx := 1;
	                initialized := TRUE;
	                output := input;
	            ELSE
	                IF clock THEN
	                    xOld := buffer[idx];
	                    buffer[idx] := input;

	                    sum := sum - xOld + input;

	                    idx := idx + 1;
	                    IF idx > windowSize THEN idx := 1; END_IF;

	                    output := sum / TO_REAL(windowSize);
	                END_IF;
	            END_IF;

	        MeanFilterType.WMA_Ramp :
	            (* Linear weights: 1..N from oldest..newest (O(1)) *)
	            IF NOT initialized THEN
	                FOR i := 1 TO windowSize DO buffer[i] := input; END_FOR;

	                denomRamp := TO_REAL(windowSize) * TO_REAL(windowSize + 1) / 2.0;

	                sum := input * TO_REAL(windowSize);
	                wsumRamp := input * denomRamp;

	                idx := 1;
	                initialized := TRUE;
	                output := input;
	            ELSE
	                IF clock THEN
	                    xOld := buffer[idx]; (* oldest *)
	                    xNew := input;

	                    sumOld := sum;

	                    buffer[idx] := xNew;

	                    (* S' = S - xOld + xNew *)
	                    sum := sumOld - xOld + xNew;

	                    (* W' = W - S_old + N*xNew *)
	                    wsumRamp := wsumRamp - sumOld + (TO_REAL(windowSize) * xNew);

	                    idx := idx + 1;
	                    IF idx > windowSize THEN idx := 1; END_IF;

	                    output := wsumRamp / denomRamp;
	                END_IF;
	            END_IF;

	        MeanFilterType.WMA_Triangular,
	        MeanFilterType.WMA_TriangularOddOnly :
	            (* Symmetric triangular weights, center-weighted (O(N)) *)
	            IF NOT initialized THEN
	                FOR i := 1 TO windowSize DO buffer[i] := input; END_FOR;
	                idx := 1;
	                initialized := TRUE;
	                output := input;
	            END_IF;

	            IF clock THEN
	                (* Update ring buffer *)
	                buffer[idx] := input;
	                idx := idx + 1;
	                IF idx > windowSize THEN idx := 1; END_IF;

	                (* Compute triangular weights *)
	                (* k=1..N from oldest..newest *)
	                mid := (windowSize + 1) / 2; (* integer div *)

	                wsumTri := 0.0;
	                denomTri := 0.0;

	                (* Oldest sample is at idx (next to overwrite) *)
	                FOR i := 0 TO windowSize - 1 DO
	                    pos := idx + i;
	                    IF pos > windowSize THEN pos := pos - windowSize; END_IF;

	                    k := i + 1;

	                    (* w = mid - |k-mid|  (triangle peak at center) *)
	                    IF k >= mid THEN
	                        dist := k - mid;
	                    ELSE
	                        dist := mid - k;
	                    END_IF;

	                    w := TO_REAL(mid - dist);
	                    wsumTri := wsumTri + w * buffer[pos];
	                    denomTri := denomTri + w;
	                END_FOR;

	                IF denomTri > 0.0 THEN
	                    output := wsumTri / denomTri;
	                ELSE
	                    output := input;
	                END_IF;
	            END_IF;

	        MeanFilterType.TRI_SMA2 :
	            (*
	             * Triangular approximation via two SMA in cascade:
	             *     y1 = SMA(input), y2 = SMA(y1). This approximates a triangular FIR well.
	            *)
	            IF NOT sma2_init THEN
	                FOR i := 1 TO windowSize DO
	                    sma2_buf1[i] := input;
	                    sma2_buf2[i] := input;
	                END_FOR;

	                sma2_sum1 := input * TO_REAL(windowSize);
	                sma2_sum2 := input * TO_REAL(windowSize);

	                sma2_idx1 := 1;
	                sma2_idx2 := 1;

	                sma2_y1 := input;
	                sma2_y2 := input;

	                sma2_init := TRUE;
	                output := input;
	            ELSE
	                IF clock THEN
	                    (* SMA stage 1 *)
	                    xOld := sma2_buf1[sma2_idx1];
	                    sma2_buf1[sma2_idx1] := input;
	                    sma2_sum1 := sma2_sum1 - xOld + input;

	                    sma2_idx1 := sma2_idx1 + 1;
	                    IF sma2_idx1 > windowSize THEN sma2_idx1 := 1; END_IF;

	                    sma2_y1 := sma2_sum1 / TO_REAL(windowSize);

	                    (* SMA stage 2 *)
	                    xOld := sma2_buf2[sma2_idx2];
	                    sma2_buf2[sma2_idx2] := sma2_y1;
	                    sma2_sum2 := sma2_sum2 - xOld + sma2_y1;

	                    sma2_idx2 := sma2_idx2 + 1;
	                    IF sma2_idx2 > windowSize THEN sma2_idx2 := 1; END_IF;

	                    sma2_y2 := sma2_sum2 / TO_REAL(windowSize);

	                    output := sma2_y2;
	                END_IF;
	            END_IF;

	        MeanFilterType.EMA :
	            (* EMA (alpha mandatory) *)
	            IF NOT initialized THEN
	                emaY := input;
	                initialized := TRUE;
	            ELSE
	                IF clock THEN
	                    emaY := emaY + emaAlpha * (input - emaY);
	                END_IF;
	            END_IF;

	            output := emaY;
	    END_CASE;

	    done := NOT error;
	ELSE
	    busy := FALSE;
	    done := FALSE;
	END_IF;
	END_FUNCTION_BLOCK

(* ---- SShapedFunc.pou ---- *)
(*#-#-#-#-#-#-#-#-#-#---Declaration---#-#-#-#-#-#-#-#-#-#-#-#-#*)

{attribute 'no_assign'}
FUNCTION_BLOCK SShapedFunc
VAR_INPUT
    execute : BOOL; (* PLCopen: Start on rising edge *)
    clock : BOOL;
    startValue : REAL;
    endValue : REAL;
    duration : TIME;
    tickTime : TIME := T#10ms;
END_VAR
VAR_OUTPUT
    output : REAL;
    done : BOOL;
    busy : BOOL;
    error : BOOL;
    errorId : INT; (* 1 : InvalidTime *)
END_VAR
VAR
    prevExecute : BOOL;
    active : BOOL;
    elapsedTicks : UDINT;
    totalTicks : UDINT;
    progress : REAL;
    deltaValue : REAL;
END_VAR

(*#-#-#-#-#-#-#-#-#-#---Implementation---#-#-#-#-#-#-#-#-#-#-#-#-#*)

(* Defaults *)
done := FALSE; busy := FALSE; error := (errorId <> 0);

(* Rising edge detection *)
IF execute AND NOT prevExecute THEN
    errorId := 0; (* Clear previous error on new rising edge *)
    (* Validate timing *)
    IF (TO_DINT(duration) <= 0) OR (TO_DINT(tickTime) <= 0) THEN
        error := TRUE;
        errorId := 1;
        active := FALSE;
    ELSE
        active := TRUE;
        elapsedTicks := 0;

        totalTicks := TO_UDINT(TO_DINT(duration) / TO_DINT(tickTime));
        IF totalTicks = 0 THEN totalTicks := 1; END_IF;

        deltaValue := endValue - startValue;
        output := startValue;
    END_IF;
END_IF;

IF execute THEN
    IF active THEN
        busy := TRUE;

        IF clock THEN
            IF elapsedTicks < totalTicks THEN
                elapsedTicks := elapsedTicks + 1;
            END_IF;
        END_IF;

        progress := TO_REAL(elapsedTicks) / TO_REAL(totalTicks);

        IF progress >= 1.0 THEN
            output := endValue;
            active := FALSE;
            done := TRUE;
        ELSE
            output := startValue + deltaValue * (3.0 * progress * progress - 2.0 * progress * progress * progress);
        END_IF;
    ELSE
        IF NOT error THEN
            done := TRUE;
        END_IF;
    END_IF;
ELSE
    (* Reset when execute is FALSE: clear state and acknowledge any error *)
    active := FALSE;
    elapsedTicks := 0;
    totalTicks := 0;
    errorId := 0;
END_IF;

prevExecute := execute;

(* ---- SShapedFunc.st ---- *)
FUNCTION_BLOCK SShapedFunc
	VAR_INPUT
	    execute : BOOL; (* PLCopen: Start on rising edge *)
	    clock : BOOL;
	    startValue : REAL;
	    endValue : REAL;
	    duration : TIME;
	    tickTime : TIME := T#10ms;
	END_VAR
	VAR_OUTPUT
	    output : REAL;
	    done : BOOL;
	    busy : BOOL;
	    error : BOOL;
	    errorId : INT; (* 1 : InvalidTime *)
	END_VAR
	VAR
	    prevExecute : BOOL;
	    active : BOOL;
	    elapsedTicks : UDINT;
	    totalTicks : UDINT;
	    progress : REAL;
	    deltaValue : REAL;
	END_VAR

	(* Defaults *)
	done := FALSE; busy := FALSE; error := (errorId <> 0);

	(* Rising edge detection *)
	IF execute AND NOT prevExecute THEN
	    errorId := 0; (* Clear previous error on new rising edge *)
	    (* Validate timing *)
	    IF (TO_DINT(duration) <= 0) OR (TO_DINT(tickTime) <= 0) THEN
	        error := TRUE;
	        errorId := 1;
	        active := FALSE;
	    ELSE
	        active := TRUE;
	        elapsedTicks := 0;

	        totalTicks := TO_UDINT(TO_DINT(duration) / TO_DINT(tickTime));
	        IF totalTicks = 0 THEN totalTicks := 1; END_IF;

	        deltaValue := endValue - startValue;
	        output := startValue;
	    END_IF;
	END_IF;

	IF execute THEN
	    IF active THEN
	        busy := TRUE;

	        IF clock THEN
	            IF elapsedTicks < totalTicks THEN
	                elapsedTicks := elapsedTicks + 1;
	            END_IF;
	        END_IF;

	        progress := TO_REAL(elapsedTicks) / TO_REAL(totalTicks);

	        IF progress >= 1.0 THEN
	            output := endValue;
	            active := FALSE;
	            done := TRUE;
	        ELSE
	            output := startValue + deltaValue * (3.0 * progress * progress - 2.0 * progress * progress * progress);
	        END_IF;
	    ELSE
	        IF NOT error THEN
	            done := TRUE;
	        END_IF;
	    END_IF;
	ELSE
	    (* Reset when execute is FALSE: clear state and acknowledge any error *)
	    active := FALSE;
	    elapsedTicks := 0;
	    totalTicks := 0;
	    errorId := 0;
	END_IF;

	prevExecute := execute;
	END_FUNCTION_BLOCK
